// TwinCAT 3 PLC project TrafficLightPLC
// ProgramVersion: 3.1.4024.0
// libraries:
//   Tc2_Standard, * (Beckhoff Automation GmbH)
//   Tc2_System, * (Beckhoff Automation GmbH)
//   Tc3_Module, * (Beckhoff Automation GmbH)
//   VisuSymbols,3.5.10.0,System
// project tree:
//   DUTs/ E_Light.TcDUT
//   / GlobalTextList.TcGTLO, PlcTask.TcTTO, Visualization Manager.TcVMO (not stored)
//   GVLs/ GVL.TcGVL
//   POUs/ FB_TrafficLight.TcPOU, FB_TrafficLightController.TcPOU, MAIN.TcPOU
//   VISUs/ visuTrafficLights.TcVIS
// real-time tasks:
//   TASK PlcTask: cycle T#10ms, priority 20, ADS port 350

CONFIGURATION TrafficLightPLC
    RESOURCE PLC ON TwinCAT3
        TASK PlcTask(INTERVAL := T#10ms, PRIORITY := 20);
        PROGRAM MAIN WITH PlcTask : MAIN;
    END_RESOURCE
END_CONFIGURATION

// ---- DUTs/E_Light.TcDUT
{attribute 'qualified_only'}
{attribute 'strict'}
TYPE E_Light :
(
	Red := 0,
	Yellow := 1,
	Green := 2
);
END_TYPE

// ---- GVLs/GVL.TcGVL
{attribute 'qualified_only'}
VAR_GLOBAL CONSTANT
	MAX_TRAFFIC_LIGHTS: SINT := 4;
END_VAR

// ---- POUs/MAIN.TcPOU
PROGRAM MAIN
VAR
	fbTrafficLightController: FB_TrafficLightController;
	nNumTraffic: SINT := 4;
	bInitialized: BOOL := FALSE;
END_VAR

IF NOT bInitialized THEN
	bInitialized := TRUE;
	Setup();
END_IF

fbTrafficLightController();

METHOD PRIVATE Setup
fbTrafficLightController.NumberOfTrafficLights := nNumTraffic;
fbTrafficLightController.Setup(2, T#10S, T#3S, T#8S);
END_METHOD

END_PROGRAM

// ---- POUs/FB_TrafficLightController.TcPOU
FUNCTION_BLOCK PUBLIC FB_TrafficLightController
VAR
	nNumberOfTrafficLights : SINT;
	currentLight: SINT := 1;
	
	arTrafficLights: ARRAY[1..4] OF FB_TrafficLight;
	arTrafficLightsInvisible: ARRAY[1..4] OF BOOL;
	
END_VAR

StartCurrentTrafficLight();

RefereshAllTrafficLights();

TrySwitchToNextTrafficLight();

PROPERTY PUBLIC NumberOfTrafficLights : SINT
GET
NumberOfTrafficLights := nNumberOfTrafficLights;
END_GET
SET
IF NumberOfTrafficLights >= 2 AND NumberOfTrafficLights <= 4 THEN
	nNumberOfTrafficLights := NumberOfTrafficLights;
	SetVisibleTrafficLights();
END_IF
END_SET
END_PROPERTY

METHOD PRIVATE RefereshAllTrafficLights
VAR
	index: SINT;
END_VAR
FOR index := 1 TO nNumberOfTrafficLights DO
	arTrafficLights[index]();
END_FOR
END_METHOD

METHOD PUBLIC Setup
VAR_INPUT
	lightNumber: SINT;
	
	redDuration: TIME;
	yellowDuration: TIME;
	greenDuration: TIME;
END_VAR
IF lightNumber >= 1 AND lightNumber <= GVL.MAX_TRAFFIC_LIGHTS THEN
	arTrafficLights[lightNumber].Setup(redDuration, yellowDuration, greenDuration);
END_IF
END_METHOD

METHOD PRIVATE SetVisibleTrafficLights
VAR
	idx: INT;
END_VAR
FOR idx := 1 TO GVL.MAX_TRAFFIC_LIGHTS DO
	arTrafficLightsInvisible[idx] := TRUE;
END_FOR

FOR idx := 1 TO nNumberOfTrafficLights DO
	arTrafficLightsInvisible[idx] := FALSE;
END_FOR
END_METHOD

METHOD PRIVATE StartCurrentTrafficLight
IF NOT arTrafficLights[currentLight].Start THEN
	arTrafficLights[currentLight].Start := TRUE;
END_IF
END_METHOD

METHOD PRIVATE TrySwitchToNextTrafficLight
IF arTrafficLights[currentLight].CanSwitch() THEN
	currentLight := currentLight + 1;
	IF currentLight > nNumberOfTrafficLights THEN
		currentLight := 1;
	END_IF
END_IF
END_METHOD

END_FUNCTION_BLOCK

// ---- POUs/FB_TrafficLight.TcPOU
FUNCTION_BLOCK PUBLIC FB_TrafficLight
VAR
	tRedDuration: TIME := T#6S;
	tYellowDuration: TIME := T#2S;
	tGreenDuration: TIME := T#4S;
	
	fbTon: TON;
	
	RedLight: BOOL;
	YellowLight: BOOL;
	GreenLight: BOOL;
	
	nStep: SINT := 0;
	bStart: BOOL := FALSE;
	bSwitach: BOOL := FALSE;
END_VAR

IF bStart THEN
	CASE nStep OF
		0: (* GREEN *)
			TurnOnLight(E_Light.Green);
			fbTon(IN := TRUE, PT := tGreenDuration);
			IF fbTon.Q THEN
				fbTon(IN := FALSE);
				nStep := 1;
			END_IF
		1: (* YELLOW *)
			TurnOnLight(E_Light.Yellow);
			fbTon(IN := TRUE, PT := tYellowDuration);
			IF fbTon.Q THEN
				fbTon(IN := FALSE);
				nStep := 2;
				bSwitach := TRUE;
			END_IF
		2: (* RED *)
			TurnOnLight(E_Light.Red);
			fbTon(IN := TRUE, PT := tRedDuration);
			IF fbTon.Q THEN
				fbTon(IN := FALSE);
				nStep := 0;
				bStart := FALSE;
			END_IF
	END_CASE
ELSE
	TurnOnLight(E_Light.Red);
END_IF

METHOD PUBLIC CanSwitch : BOOL
VAR
	bReturn: BOOL := FALSE;
END_VAR
IF bSwitach THEN
	bReturn := TRUE;
	bSwitach := FALSE;
END_IF
CanSwitch := bReturn;
END_METHOD

METHOD PUBLIC Setup
VAR_INPUT
	redDuration: TIME;
	yellowDuration: TIME;
	greenDuration: TIME;
END_VAR
tRedDuration := redDuration;
tYellowDuration := yellowDuration;
tGreenDuration := greenDuration;
END_METHOD

PROPERTY PUBLIC Start : BOOL
GET
Start := bStart;
END_GET
SET
bStart := Start;
END_SET
END_PROPERTY

METHOD PRIVATE TurnOnLight
VAR_INPUT
	eLight: E_Light;
END_VAR
CASE eLight OF
	E_Light.Red:
		IF NOT RedLight THEN
			RedLight := TRUE;
			YellowLight := FALSE;
			GreenLight := FALSE;
		END_IF 

	E_Light.Yellow:
		IF NOT YellowLight THEN
			RedLight := FALSE;
			YellowLight := TRUE;
			GreenLight := FALSE;
		END_IF 

	
	E_Light.Green:
		IF NOT GreenLight THEN
			RedLight := FALSE;
			YellowLight := FALSE;
			GreenLight := TRUE;
		END_IF 

	ELSE
		RedLight := FALSE;
		YellowLight := FALSE;
		GreenLight := FALSE;
END_CASE
END_METHOD

END_FUNCTION_BLOCK

// ---- VISUs/visuTrafficLights.TcVIS
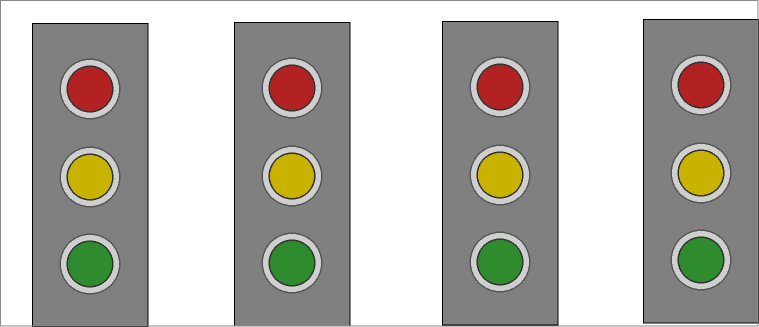
VISUALIZATION visuTrafficLights  // 759x327
    RoundedRectangle (32,23 116x304), invisible if: MAIN.fbTrafficLightController.arTrafficLightsInvisible[1]
    Lamp1 (55,54 70x70), variable: MAIN.fbTrafficLightController.arTrafficLights[1].RedLight, invisible if: MAIN.fbTrafficLightController.arTrafficLightsInvisible[1], style: Lamp-Lamp1-Red
    Lamp1 (55,142 70x70), variable: MAIN.fbTrafficLightController.arTrafficLights[1].YellowLight, invisible if: MAIN.fbTrafficLightController.arTrafficLightsInvisible[1], style: Lamp-Lamp1-Yellow
    Lamp1 (55,229 70x70), variable: MAIN.fbTrafficLightController.arTrafficLights[1].GreenLight, invisible if: MAIN.fbTrafficLightController.arTrafficLightsInvisible[1], style: Lamp-Lamp1-Green
    RoundedRectangle (234,22 116x304), invisible if: MAIN.fbTrafficLightController.arTrafficLightsInvisible[2]
    Lamp1 (257,53 70x70), variable: MAIN.fbTrafficLightController.arTrafficLights[2].RedLight, invisible if: MAIN.fbTrafficLightController.arTrafficLightsInvisible[2], style: Lamp-Lamp1-Red
    Lamp1 (257,141 70x70), variable: MAIN.fbTrafficLightController.arTrafficLights[2].YellowLight, invisible if: MAIN.fbTrafficLightController.arTrafficLightsInvisible[2], style: Lamp-Lamp1-Yellow
    Lamp1 (257,228 70x70), variable: MAIN.fbTrafficLightController.arTrafficLights[2].GreenLight, invisible if: MAIN.fbTrafficLightController.arTrafficLightsInvisible[2], style: Lamp-Lamp1-Green
    RoundedRectangle (442,21 116x304), invisible if: MAIN.fbTrafficLightController.arTrafficLightsInvisible[3]
    Lamp1 (465,52 70x70), variable: MAIN.fbTrafficLightController.arTrafficLights[3].RedLight, invisible if: MAIN.fbTrafficLightController.arTrafficLightsInvisible[3], style: Lamp-Lamp1-Red
    Lamp1 (465,140 70x70), variable: MAIN.fbTrafficLightController.arTrafficLights[3].YellowLight, invisible if: MAIN.fbTrafficLightController.arTrafficLightsInvisible[3], style: Lamp-Lamp1-Yellow
    Lamp1 (465,227 70x70), variable: MAIN.fbTrafficLightController.arTrafficLights[3].GreenLight, invisible if: MAIN.fbTrafficLightController.arTrafficLightsInvisible[3], style: Lamp-Lamp1-Green
    RoundedRectangle (643,19 116x304), invisible if: MAIN.fbTrafficLightController.arTrafficLightsInvisible[4]
    Lamp1 (666,50 70x70), variable: MAIN.fbTrafficLightController.arTrafficLights[4].RedLight, invisible if: MAIN.fbTrafficLightController.arTrafficLightsInvisible[4], style: Lamp-Lamp1-Red
    Lamp1 (666,138 70x70), variable: MAIN.fbTrafficLightController.arTrafficLights[4].YellowLight, invisible if: MAIN.fbTrafficLightController.arTrafficLightsInvisible[4], style: Lamp-Lamp1-Yellow
    Lamp1 (666,225 70x70), variable: MAIN.fbTrafficLightController.arTrafficLights[4].GreenLight, invisible if: MAIN.fbTrafficLightController.arTrafficLightsInvisible[4], style: Lamp-Lamp1-Green
END_VISUALIZATION
